TYPE SafetyEmergencyStopsProcesses :
STRUCT
	///Reset the errors (including the programmed ones and the TwinSAFE group ones)
	reset: Process;
END_STRUCT
END_TYPE

(* stored: Version 1.1.0.1, ProductVersion 3.1.4019.2
   DUT SafetyEmergencyStopsProcesses: Id {4b053688-05aa-4882-8b10-73ee54b10e9e} *)
